{region '#Template'}
	{attribute 'Version' := '5.0.0.0'}
	{attribute 'Tags' := '"LCID": "1031", "Text": "Fassade, Sonnenschutz, Wartung"'}
	{attribute 'Tags' := '"LCID": "1033", "Text": "Facade, Sunprotection, Maintenance"'}
	{attribute 'Using' := '"Type": "Template", "URI": "ST_BA_SunBld"'}
	{attribute 'Using' := '"Type": "Template", "URI": "E_BA_SunBldPrio"'}
	{attribute 'Description' := '"LCID": "1031", "Text": "Sonnenschutz Wartungsposition"'}
	{attribute 'Description' := '"LCID": "1033", "Text": "Sunprotection maintenance-position"'}
{endregion}
FUNCTION_BLOCK FB_BA_Facade_Maintenance EXTENDS FB_BA_View
VAR_INPUT
END_VAR
VAR_OUTPUT
	stSunBld		: ST_BA_SunBld;
	bMntnActv		: BOOL;
END_VAR
VAR_INPUT CONSTANT
	MntnEn			: FB_BA_BV_Op;		
	MntnPos			: FB_BA_AV_Op;		
	MntnAngl		: FB_BA_AV_Op;
	MntnEvent		: FB_BA_SunBldEvt := (ePrio:=E_BA_SunBldPrio.eMaintenance);			
END_VAR
VAR
END_VAR

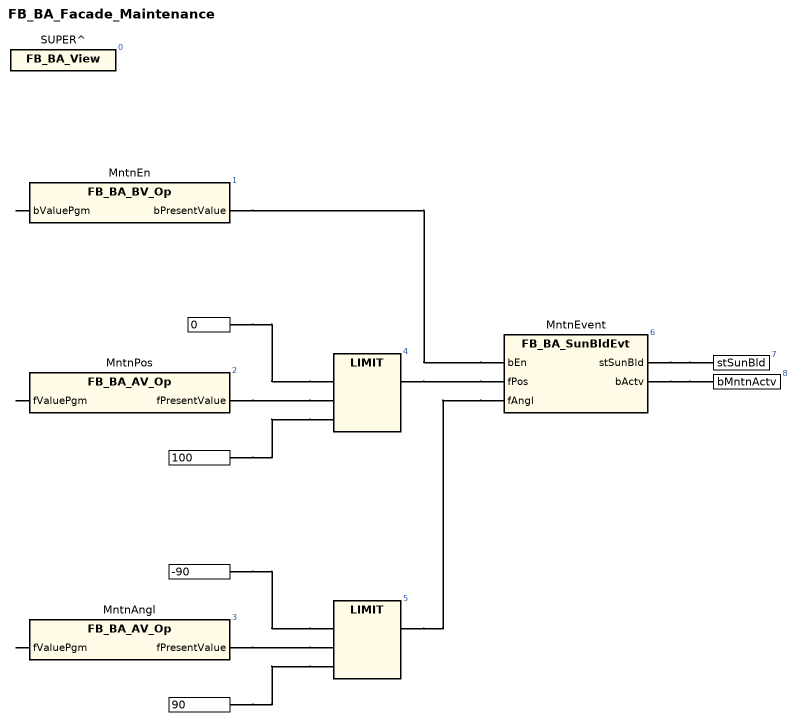
SUPER^(); // FB_BA_View
MntnEn(); // FB_BA_BV_Op
MntnPos(); // FB_BA_AV_Op
MntnAngl(); // FB_BA_AV_Op
MntnEvent(
    bEn := MntnEn.bPresentValue,
    fPos := LIMIT(0, MntnPos.fPresentValue, 100),
    fAngl := LIMIT(-90, MntnAngl.fPresentValue, 90)); // FB_BA_SunBldEvt
stSunBld := MntnEvent.stSunBld;
bMntnActv := MntnEvent.bActv;

METHOD FB_init : BOOL
VAR_INPUT
	bInitRetains : BOOL; // if TRUE; the retain variables are initialized (warm start / cold start)
	bInCopyCode : BOOL;  // if TRUE; the instance afterwards gets moved into the copy code (online change)
END_VAR
MntnEn.iParent					:= THIS^;
MntnEn.iLabel					:= LblCtl_MaintenanceEnable;
MntnEn.sObjectName		   		:= '{Idx=01}';
MntnEn.sInactiveText			:= txtEvent_Off;
MntnEn.sActiveText				:= txtEvent_On;
MntnEn.bValueRm					:= FALSE;
MntnEn.eToggleMode				:= E_BA_ToggleMode.eSwitch;        
                            	                   	
MntnPos.iParent					:= THIS^;
MntnPos.iLabel					:= LblCtl_MaintenancePosition;
MntnPos.sObjectName		   		:= '{Idx=01}';
MntnPos.eUnit					:= E_BA_Unit.eOther_Percent; 
MntnPos.fValueRm				:= 0.0;
                            	
		                    	
MntnAngl.iParent				:= THIS^;
MntnAngl.iLabel					:= LblCtl_MaintenanceAngle;	
MntnAngl.sObjectName		   	:= '{Idx=02}';
MntnAngl.eUnit					:= E_BA_Unit.eOther_DegreesAngular; 
MntnAngl.fValueRm				:= 0.0;
END_METHOD

END_FUNCTION_BLOCK

(* stored: Version 1.1.0.1, ProductVersion 3.1.4024.12
   POU FB_BA_Facade_Maintenance: Id {0e2c0dd9-fd99-4563-b608-a4fe81cf476a}, SpecialFunc None
   Method FB_init: Id {cd74ee3d-2069-4954-b66e-6487e9b05302} *)
